// TIA Portal V17 export
// export: Created 2024-09-02T12:50:34.7141059Z, ExportSetting WithDefaults, DisplayName Totally Integrated Automation Portal, DisplayVersion V17, DisplayName TIA Portal Openness, DisplayVersion V17, DisplayName TIA Portal Version Control Interface, DisplayVersion V17, DisplayName STEP 7 Professional, DisplayVersion V17, DisplayName STEP 7 Safety, DisplayVersion V17, DisplayName WinCC Professional, DisplayVersion V17
TYPE "typ_AnbauteilVorg"
// stored: IsFailsafeCompliant false
   STRUCT
      Bauteil { S7_SetPoint := 'True'} : "typ_Anbauteil";   // Scancode Bauteil Soll / Scancode Component Target
      Alternativ_1 { S7_SetPoint := 'True'} : "typ_Anbauteil";   // Scancode Alternativ 1 Bauteil Soll / Scancode Alternative 1 Component Target
      Alternativ_2 { S7_SetPoint := 'True'} : "typ_Anbauteil";   // Scancode Alternativ 2 Bauteil Soll / Scancode Alternative 2 Component Target
      Reserve : String[76];   // Reserve
   END_STRUCT;
END_TYPE
